{attribute 'call_after_init'}
FUNCTION_BLOCK FINAL _SYS_COMP_FirstObject EXTENDS Object
VAR_INPUT
END_VAR
VAR_OUTPUT
END_VAR
VAR
END_VAR

END_FUNCTION_BLOCK

(* stored: Version 1.1.0.1, ProductVersion 3.1.4024.12
   POU _SYS_COMP_FirstObject: Id {c51e1415-84bf-474c-b3c8-ec8737582e96}, SpecialFunc None *)
